TYPE LoopIterator : INT; END_TYPE

(* stored: Version 1.1.0.1, ProductVersion 3.1.4024.10
   DUT LoopIterator: Id {c895961f-2bac-4da7-ba9f-e3ff4e9d4be9} *)
